PROGRAM P_Demo_FB_DMXGetDeviceInfo
VAR
    fbGetDeviceInfo   : FB_DMXGetDeviceInfo;          // 读设备综合信息
    stDmxCmdBuffer    : ST_DMXCommandBuffer;          // 与通讯 FB 共用
    wTargetManufId    : WORD := 16#4241;              // 目标灯具厂商 ID
    dwTargetDeviceId  : DWORD := 16#12131415;         // 目标灯具设备 ID
    byTargetPort      : BYTE := 0;                    // 根设备通道 0
    bDoRead           : BOOL := FALSE;                // 在线给一次上升沿触发
    bBusy             : BOOL;
    bError            : BOOL;
    udiErrId          : UDINT;
    stDeviceInfo      : ST_DMXDeviceInfo;             // 设备综合信息
END_VAR

// ============================================================
// Tc2_DMX.FB_DMXGetDeviceInfo 演示程序
// ============================================================
// 场景：接入陌生第三方灯具时先读 DEVICE_INFO 摸清型号、协议版本、占用通道数、子设备/传感器情况。
// 价值：一次调用拿到设备全貌，免去逐个 PID 试探，是设备接入/自检流程的起点。
// 验证：给 bDoRead 一次上升沿 -> bBusy 短暂 TRUE -> 回 FALSE 后 stDeviceInfo 各字段（如 DMX512 占用槽数、子设备数）有值；设备不在线则 bError 且 udiErrId=0x8002。
// 验证步骤：
//   1. 右键 PLC 项目下 POUs 文件夹 → Add → Existing Item → 选本 .TcPOU 文件
//   2. 引用 Tc2_DMX；同项目里放一个 FB_EL6851CommunicationEx 实例并共用 stDmxCmdBuffer（非 CycleMode）
//   3. 编译 → 登录 → 运行；按上方『验证』行在线给上升沿观察
// ============================================================

fbGetDeviceInfo(
    bStart                     := bDoRead,
    wDestinationManufacturerId := wTargetManufId,
    dwDestinationDeviceId      := dwTargetDeviceId,
    byPortId                   := byTargetPort,
    dwOptions                  := 0,
    stCommandBuffer            := stDmxCmdBuffer,
    bBusy                      => bBusy,
    bError                     => bError,
    udiErrorId                 => udiErrId,
    stDMXDeviceInfo            => stDeviceInfo
);

END_PROGRAM

(* stored: Version 1.1.0.1, ProductVersion 3.1.4024.5
   POU P_Demo_FB_DMXGetDeviceInfo: Id {551d11e7-eecf-596d-b3aa-eac3e1bd0752}, SpecialFunc None *)
